// TIA Portal V20 export
TYPE "TypeWenglorP3PC301Rd"
   STRUCT
      Measure : DInt;   // Actual measured value 60.000...66000µm (-1= Read error)
      Scale : SInt;   // Scale -6 = µm
      SCC1 : Bool;   // Signal output 1 (1= Occ)
      SCC2 : Bool;   // Signal output 2 (1= Occ)
      Err : Bool;   // Signal sensor error (1= Error)
      Warn : Bool;   // Signal sensor warning(1= warning)
      Warn1 : Bool;   // Indication Error / Warning (1= true)
      Warn2 : Bool;   // Indication Error / Warning (1= true)
      Warn3 : Bool;   // Indication Error / Warning (1= true)
      Warn4 : Bool;   // Indication Error / Warning (1= true)
   END_STRUCT;
END_TYPE
